FUNCTION_BLOCK PRG_GEM1
VAR_INPUT
END_VAR
VAR_OUTPUT
END_VAR
VAR
END_VAR

END_FUNCTION_BLOCK

(* stored: Version 1.1.0.1, ProductVersion 3.1.4022.16
   POU PRG_GEM1: Id {b5aed3c6-13be-428f-86ce-8bd830676022}, SpecialFunc None *)
